// TIA Portal V20 export
TYPE "UDT_RecepcionDeMesa"
   STRUCT
      Auxiliar_01 : UInt;
      MesaSalidaMultiDestino : UInt;
      Auxiliar_03 : UInt;
      Auxiliar_04 : UInt;
      Protocolo { S7_SetPoint := 'True'} : "UDT_ProtocoloRecMesa";
   END_STRUCT;
END_TYPE
